PROGRAM IntervaloLavCalibr
VAR PERSISTENT
	IntervaloLavagem	:UDINT;	//Intervalo entre lavagens - Vem da IHM (h)
	AlarmeLavagem		:BOOL;	//Alguma linha excedeu o tempo de lavagem
	LinhaLavagem		:INT;	//Linha que excedeu o tempo de lavagem
	
	IntervaloCalibracao	:UDINT;	//Intervalo entre calibrações - Vem da IHM (h)
	AlarmeCalibracao	:BOOL;	//Alguma linha excedeu o tempo de calibração
	LinhaCalibracao		:INT;	//Linha que excedeu o tempo de calibração
	
END_VAR

VAR
	
	teste:LINT;
	teste2:LINT;
	TOF_Alarme: TOF;
	TOF_Calibracao: TOF;
END_VAR

//Essa rotina verifica se alguma calibração ou lavagem excedeu o tempo definido, subindo um alarme na IHM

//Verifica se alguma linha escedeu o intervalo entre lavagens. A primeira detectada, gera um alarme na IHM
TOF_Alarme(IN:= AlarmeLavagem, PT:= T#1S, Q=> , ET=> );	//Temporizador para garantir que a IHM conseguirá detectar a borda de subida do alarme
TOF_Calibracao(IN:= AlarmeCalibracao, PT:= T#1S, Q=> , ET=> );	//Temporizador para garantir que a IHM conseguirá detectar a borda de subida do alarme

{Region "Alarmes da lavagem}
	AlarmeLavagem := FALSE;	//Inicia a variável
	IF (DT_TO_LINT(Main.HoraAtual) - Liquidos.UltimoAlrLavagem[1]) > IntervaloLavagem * 3600 THEN
		Liquidos.UltimoAlrLavagem[1] := DT_TO_LINT(Main.HoraAtual) + (IntervaloLavagem * 360); 
		AlarmeLavagem := TRUE;
		LinhaLavagem := 1;
			
	ELSIF (DT_TO_LINT(Main.HoraAtual) - Liquidos.UltimoAlrLavagem[2]) > IntervaloLavagem * 3600 THEN
		Liquidos.UltimoAlrLavagem[2] := DT_TO_LINT(Main.HoraAtual) + (IntervaloLavagem * 360);
		AlarmeLavagem := TRUE;
		LinhaLavagem := 2;	
			
	ELSIF (DT_TO_LINT(Main.HoraAtual) - Liquidos.UltimoAlrLavagem[3]) > IntervaloLavagem * 3600 THEN
		Liquidos.UltimoAlrLavagem[3] := DT_TO_LINT(Main.HoraAtual) + (IntervaloLavagem * 360);
		AlarmeLavagem := TRUE;
		LinhaLavagem := 3;	
			
	ELSIF (DT_TO_LINT(Main.HoraAtual) - Liquidos.UltimoAlrLavagem[4]) > IntervaloLavagem * 3600 THEN
		Liquidos.UltimoAlrLavagem[4] := DT_TO_LINT(Main.HoraAtual) + (IntervaloLavagem * 360);
		AlarmeLavagem := TRUE;
		LinhaLavagem := 4;	
			
	ELSIF (DT_TO_LINT(Main.HoraAtual) - Liquidos.UltimoAlrLavagem[5]) > IntervaloLavagem * 3600 THEN
		Liquidos.UltimoAlrLavagem[5] := DT_TO_LINT(Main.HoraAtual) + (IntervaloLavagem * 360);
		AlarmeLavagem := TRUE;
		LinhaLavagem := 5;	
			
	ELSIF (DT_TO_LINT(Main.HoraAtual) - Liquidos.UltimoAlrLavagem[6]) > IntervaloLavagem * 3600 THEN
		Liquidos.UltimoAlrLavagem[6] := DT_TO_LINT(Main.HoraAtual) + (IntervaloLavagem * 360);
		AlarmeLavagem := TRUE;
		LinhaLavagem := 6;	
			
	ELSIF (DT_TO_UDINT(Main.HoraAtual) - Liquidos.UltimoAlrLavagem[7]) > IntervaloLavagem * 3600 THEN
		Liquidos.UltimoAlrLavagem[7] := DT_TO_LINT(Main.HoraAtual) + (IntervaloLavagem * 360);
		AlarmeLavagem := TRUE;
		LinhaLavagem := 7;	
			
	ELSIF (DT_TO_UDINT(Main.HoraAtual) - Liquidos.UltimoAlrLavagem[8]) > IntervaloLavagem * 3600 THEN
		Liquidos.UltimoAlrLavagem[8] := DT_TO_LINT(Main.HoraAtual) + (IntervaloLavagem * 360);
		AlarmeLavagem := TRUE;
		LinhaLavagem := 8;	
			
	ELSIF (DT_TO_LINT(Main.HoraAtual) - Liquidos.UltimoAlrLavagem[9]) > IntervaloLavagem * 3600 THEN
		Liquidos.UltimoAlrLavagem[9] := DT_TO_LINT(Main.HoraAtual) + (IntervaloLavagem * 360);
		AlarmeLavagem := TRUE;
		LinhaLavagem := 9;	
			
	ELSIF (DT_TO_LINT(Main.HoraAtual) - Liquidos.UltimoAlrLavagem[10]) > IntervaloLavagem * 3600 THEN
		Liquidos.UltimoAlrLavagem[10] := DT_TO_LINT(Main.HoraAtual) + (IntervaloLavagem * 360);
		AlarmeLavagem := TRUE;
		LinhaLavagem := 10;	
			
	ELSIF (DT_TO_LINT(Main.HoraAtual) - Liquidos.UltimoAlrLavagem[11]) > IntervaloLavagem * 3600 THEN
		Liquidos.UltimoAlrLavagem[11] := DT_TO_LINT(Main.HoraAtual) + (IntervaloLavagem * 360);
		AlarmeLavagem := TRUE;
		LinhaLavagem := 11;
				
	ELSIF (DT_TO_LINT(Main.HoraAtual) - Liquidos.UltimoAlrLavagem[12]) > IntervaloLavagem * 3600 THEN
		Liquidos.UltimoAlrLavagem[12] := DT_TO_LINT(Main.HoraAtual) + (IntervaloLavagem * 360);
		AlarmeLavagem := TRUE;
		LinhaLavagem := 12;
	END_IF
{endregion}

teste2 := DT_TO_LINT(Main.HoraAtual);
teste := (DT_TO_LINT(Main.HoraAtual) - HMI.UltimoAlrCalibr[1]);
{Region "Alarmes da calibração"}
	AlarmeCalibracao := FALSE;
	IF DT_TO_UDINT(Main.HoraAtual) - HMI.UltimoAlrCalibr[1] > IntervaloCalibracao * 3600 THEN
		HMI.UltimoAlrCalibr[1] := DT_TO_LINT(Main.HoraAtual) + (IntervaloCalibracao * 360);	//Se o alarme subir e a linha não for calibrada, o alarme subirá após 1/10 do intervalo
		AlarmeCalibracao := TRUE;
		LinhaCalibracao := 1;
	ELSIF DT_TO_UDINT(Main.HoraAtual) - HMI.UltimoAlrCalibr[2] > IntervaloCalibracao * 3600 THEN
		HMI.UltimoAlrCalibr[2] := DT_TO_LINT(Main.HoraAtual) + (IntervaloCalibracao * 360);	//Se o alarme subir e a linha não for calibrada, o alarme subirá após 1/10 do intervalo
		AlarmeCalibracao := TRUE;
		LinhaCalibracao := 2;
	ELSIF DT_TO_UDINT(Main.HoraAtual) - HMI.UltimoAlrCalibr[3] > IntervaloCalibracao * 3600 THEN
		HMI.UltimoAlrCalibr[3] := DT_TO_LINT(Main.HoraAtual) + (IntervaloCalibracao * 360);	//Se o alarme subir e a linha não for calibrada, o alarme subirá após 1/10 do intervalo
		AlarmeCalibracao := TRUE;
		LinhaCalibracao := 3;
	ELSIF DT_TO_UDINT(Main.HoraAtual) - HMI.UltimoAlrCalibr[4] > IntervaloCalibracao * 3600 THEN
		HMI.UltimoAlrCalibr[4] := DT_TO_LINT(Main.HoraAtual) + (IntervaloCalibracao * 360);	//Se o alarme subir e a linha não for calibrada, o alarme subirá após 1/10 do intervalo
		AlarmeCalibracao := TRUE;
		LinhaCalibracao := 4;
	ELSIF DT_TO_UDINT(Main.HoraAtual) - HMI.UltimoAlrCalibr[5] > IntervaloCalibracao * 3600 THEN
		HMI.UltimoAlrCalibr[5] := DT_TO_LINT(Main.HoraAtual) + (IntervaloCalibracao * 360);	//Se o alarme subir e a linha não for calibrada, o alarme subirá após 1/10 do intervalo
		AlarmeCalibracao := TRUE;
		LinhaCalibracao := 5;
	ELSIF DT_TO_UDINT(Main.HoraAtual) - HMI.UltimoAlrCalibr[6] > IntervaloCalibracao * 3600 THEN
		HMI.UltimoAlrCalibr[6] := DT_TO_LINT(Main.HoraAtual) + (IntervaloCalibracao * 360);	//Se o alarme subir e a linha não for calibrada, o alarme subirá após 1/10 do intervalo
		AlarmeCalibracao := TRUE;
		LinhaCalibracao := 6;
	ELSIF DT_TO_UDINT(Main.HoraAtual) - HMI.UltimoAlrCalibr[7] > IntervaloCalibracao * 3600 THEN
		HMI.UltimoAlrCalibr[7] := DT_TO_LINT(Main.HoraAtual) + (IntervaloCalibracao * 360);	//Se o alarme subir e a linha não for calibrada, o alarme subirá após 1/10 do intervalo
		AlarmeCalibracao := TRUE;
		LinhaCalibracao := 7;
	ELSIF DT_TO_UDINT(Main.HoraAtual) - HMI.UltimoAlrCalibr[8] > IntervaloCalibracao * 3600 THEN
		HMI.UltimoAlrCalibr[8] := DT_TO_LINT(Main.HoraAtual) + (IntervaloCalibracao * 360);	//Se o alarme subir e a linha não for calibrada, o alarme subirá após 1/10 do intervalo
		AlarmeCalibracao := TRUE;
		LinhaCalibracao := 8;
	ELSIF DT_TO_UDINT(Main.HoraAtual) - HMI.UltimoAlrCalibr[9] > IntervaloCalibracao * 3600 THEN
		HMI.UltimoAlrCalibr[9] := DT_TO_LINT(Main.HoraAtual) + (IntervaloCalibracao * 360);	//Se o alarme subir e a linha não for calibrada, o alarme subirá após 1/10 do intervalo
		AlarmeCalibracao := TRUE;
		LinhaCalibracao := 9;
	ELSIF DT_TO_UDINT(Main.HoraAtual) - HMI.UltimoAlrCalibr[10] > IntervaloCalibracao * 3600 THEN
		HMI.UltimoAlrCalibr[10] := DT_TO_LINT(Main.HoraAtual) + (IntervaloCalibracao * 360);	//Se o alarme subir e a linha não for calibrada, o alarme subirá após 1/10 do intervalo
		AlarmeCalibracao := TRUE;
		LinhaCalibracao := 10;
	ELSIF DT_TO_UDINT(Main.HoraAtual) - HMI.UltimoAlrCalibr[11] > IntervaloCalibracao * 3600 THEN
		HMI.UltimoAlrCalibr[11] := DT_TO_LINT(Main.HoraAtual) + (IntervaloCalibracao * 360);	//Se o alarme subir e a linha não for calibrada, o alarme subirá após 1/10 do intervalo
		AlarmeCalibracao := TRUE;
		LinhaCalibracao := 11;
	ELSIF DT_TO_UDINT(Main.HoraAtual) - HMI.UltimoAlrCalibr[12] > IntervaloCalibracao * 3600 THEN
		HMI.UltimoAlrCalibr[12] := DT_TO_LINT(Main.HoraAtual) + (IntervaloCalibracao * 360);	//Se o alarme subir e a linha não for calibrada, o alarme subirá após 1/10 do intervalo
		AlarmeCalibracao := TRUE;
		LinhaCalibracao := 12;
	END_IF
{endregion}

END_PROGRAM

(* stored: Version 1.1.0.1, ProductVersion 3.1.4024.14
   POU IntervaloLavCalibr: Id {25666d94-579e-4ac7-a152-c4150ffbbcf1}, SpecialFunc None *)
